Omron CX-Programmer project NewProject (CX-Programmer 9.61)

# PLC NewPLC1: CP1H X

## Global symbols (name address type ; comment)
0.00 BOOL  ; LIN3_FW
0.01 BOOL  ; EMG
0.02 BOOL  ; SY1
0.03 BOOL  ; CY1_FW
0.04 BOOL  ; CY1_BW
0.05 BOOL  ; CY2_A_1_BW
0.06 BOOL  ; CY2_A_2_BW
0.07 BOOL  ; CY3_FW
0.08 BOOL  ; CY3_BW
0.09 BOOL  ; CY4_A_1_BW
0.10 BOOL  ; CY4_A_2_BW
0.11 BOOL  ; S1_GRIPPER
100.00 BOOL  ; 1Y1
100.01 BOOL  ; 1Y2
100.02 BOOL  ; 2Y1
100.03 BOOL  ; 2Y2
100.04 BOOL  ; 4Y1
100.05 BOOL  ; 4Y2
100.06 BOOL  ; 3Y1
100.07 BOOL  ; 3Y2
101.00 BOOL  ; buzzzer
101.01 BOOL  ; ACTIVATE_SMC
101.02 BOOL  ; TRIGGER_MC2
101.03 BOOL  ; L_RED
101.04 BOOL  ; MOTOR_CONVEYOR
101.05 BOOL  ; TRIGGER RELAY
101.06 BOOL  ; ACTIVATE_MC2
102.00 BOOL  ; IN0 L1
102.01 BOOL  ; IN1 L1
102.02 BOOL  ; IN2 L1
102.03 BOOL  ; SETUP L1
102.04 BOOL  ; HOLD L1
102.05 BOOL  ; DRIVE L1
102.06 BOOL  ; RESET L1
102.07 BOOL  ; SVON L1
103.00 BOOL  ; IN0 L3
103.01 BOOL  ; IN1 L3
103.02 BOOL  ; IN2 L3
103.03 BOOL  ; SETUP L3
103.04 BOOL  ; HOLD L3
103.05 BOOL  ; DRIVE L3
103.06 BOOL  ; RESET L3
103.07 BOOL  ; SVON L3
104.00 BOOL  ; IN0 L2
104.01 BOOL  ; IN1 L2
104.02 BOOL  ; IN2 L2
104.03 BOOL  ; SETUP L2
104.04 BOOL  ; HOLD L2
104.05 BOOL  ; DRIVE L2
104.06 BOOL  ; RESET L2
104.07 BOOL  ; SVON L2
105.00 BOOL  ; C1
1500.00 BOOL  ; memory
1.00 BOOL  ; SL_LOADING
1.01 BOOL  ; SUL_UNLOADING
1.02 BOOL  ; LIN2_FW
1.03 BOOL  ; LIN3_BW
1.04 BOOL  ; LIN1_FW
1.05 BOOL  ; START1_CONV
1.06 BOOL  ; START2_CONV
1.07 BOOL  ; EMG_CONV
1.08 BOOL  ; SENSOR_CONV
1.09 BOOL  ; S2_GRIPPER
2000.00 BOOL  ; STEP0
2000.01 BOOL  ; STEP1
2000.02 BOOL  ; STEP2
2000.03 BOOL  ; STEP3
2000.04 BOOL  ; STEP4
2000.05 BOOL  ; STEP5
2000.06 BOOL  ; STEP6
2000.07 BOOL  ; STEP7
2000.08 BOOL  ; STEP8
2000.09 BOOL  ; STEP9
2000.10 BOOL  ; STEP10
2000.11 BOOL  ; STEP11
2000.12 BOOL  ; STEP12
2000.13 BOOL  ; STEP13
2000.14 BOOL  ; STEP14
2000.15 BOOL  ; STEP15
2001.00 BOOL  ; STEP1_2
2002.00 BOOL  ; STEP16
2002.01 BOOL  ; STEP17
2002.02 BOOL  ; STEP18
2002.03 BOOL  ; STEP19
2002.04 BOOL  ; STEP20
200.01 BOOL  ; HMI-PON
200.02 BOOL  ; HMI-POFF
200.03 BOOL  ; HMI-INIT
200.06 BOOL  ; START SIG AUTO
200.07 BOOL  ; STOP SIG AUTO
200.10 BOOL  ; fast
200.11 BOOL  ; RESET_LINEAR
201.00 BOOL  ; LIN_ON
201.01 BOOL  ; INIT LIN1
201.02 BOOL  ; LIN EMG OK
201.03 BOOL  ; LIN_ALM_OK
201.04 BOOL  ; INIT LIN2
201.05 BOOL  ; INIT LIN3
201.06 BOOL  ; INIT_CYL
201.07 BOOL  ; CYL_GRIP_INPOS
201.08 BOOL  ; CYL3_INPOS
201.09 BOOL  ; CYL1_INPOS
201.10 BOOL  ; INIT_CYL)OK
201.11 BOOL  ; INIT LIN OK
201.12 BOOL  ; Trigger_Auto
201.13 BOOL  ; AUTOSIG
201.14 BOOL  ; INIT OK
202.00 BOOL  ; LIN_1_Forward
202.01 BOOL  ; LIN_1_Backward
22.15 BOOL  ; MAIN_OK
2.00 BOOL  ; OUT1_L1
2.01 BOOL  ; OUT2_L1
2.02 BOOL  ; BUSY_L1
2.03 BOOL  ; SETON_L1
2.04 BOOL  ; INP_L1
2.05 BOOL  ; SVRE_L1
2.06 BOOL  ; ESTOP_L1
2.07 BOOL  ; ALARM_L1
3000.00 BOOL  ; STEP0
3000.01 BOOL  ; STEP1
3000.02 BOOL  ; STEP2
3000.03 BOOL  ; STEP3
3000.04 BOOL  ; STEP4
3000.05 BOOL  ; STEP5
3000.06 BOOL  ; STEP6
3000.07 BOOL  ; STEP7
3000.08 BOOL  ; STEP8
3000.09 BOOL  ; STEP9
3000.10 BOOL  ; STEP10
3000.11 BOOL  ; STEP11
300.00 BOOL  ; L1_LW
300.01 BOOL  ; L2 FW
300.02 BOOL  ; L3_FW1
300.03 BOOL  ; L3_FW2
300.04 BOOL  ; MAN_CY1_FW
300.05 BOOL  ; MAN_CY2_FW
300.06 BOOL  ; MAN_CY3_FW
300.07 BOOL  ; MAN_CY4_FW
300.08 BOOL  ; L1_MAN_BW
300.11 BOOL  ; L1_MAN_FW
30.00 BOOL  ; TIM_CONV
30.01 BOOL  ; LOCK_TIM
330.00 BOOL  ; MAN_L1_P1
330.01 BOOL  ; MAN_L1_P2
330.02 BOOL  ; MAN_L2_P1
330.03 BOOL  ; MAN_L2_P2
330.04 BOOL  ; MAN_L1_P1
330.05 BOOL  ; MAN_L1_P2
350.14 BOOL  ; Alarm_EMG
350.15 BOOL  ; Alarm_Main_Air_Supply
351.00 BOOL  ; Alarm_Lin1_OFF
351.01 BOOL  ; Alarm_Lin3_OFF
351.02 BOOL  ; Alarm_Lin2_OFF
351.03 BOOL  ; Alarm_SMC1
351.04 BOOL  ; Alarm_SMC3
351.05 BOOL  ; Alarm_SMC2
3.00 BOOL  ; OUT1_L3
3.01 BOOL  ; OUT2_L3
3.02 BOOL  ; BUSY_L3
3.03 BOOL  ; SETON_L3
3.04 BOOL  ; INP_L3
3.05 BOOL  ; SVRE_L3
3.06 BOOL  ; ESTOP_L3
3.07 BOOL  ; ALARM_L3
4000.00 BOOL  ; STEP0
4000.01 BOOL  ; STEP1
4000.02 BOOL  ; STEP2
4000.03 BOOL  ; STEP3
4000.04 BOOL  ; picking_alert
400.02 BOOL  ; Timer_homing
4.00 BOOL  ; OUT1_L2
4.01 BOOL  ; OUT2_L2
4.02 BOOL  ; BUSY_L2
4.03 BOOL  ; SETON_L2
4.04 BOOL  ; INPT_L2
4.05 BOOL  ; SVRE_L2
4.06 BOOL  ; ESTOP_L2
4.07 BOOL  ; ALARM_L2
600.00 BOOL  ; L1_BW
600.01 BOOL  ; LW_BW
600.02 BOOL  ; L3_BW
600.03 BOOL  ; CY1_BW
600.04 BOOL  ; MAN_CY1_BW
600.05 BOOL  ; MAN_CY2_BW
600.06 BOOL  ; MAN_CY3_BW
600.07 BOOL  ; MAN_CY4_BW
60.00 BOOL  ; DIFD_BUSY_L1
60.01 BOOL  ; DIFD_BUSY_L3
60.02 BOOL  ; DIFD_BUSY_L2
60.03 BOOL  ; DIFU_BUSY_L1
60.04 BOOL  ; DIFU_BUSY_L3
60.05 BOOL  ; DIFU_BUSY_L2
700.00 BOOL  ; L1 MAN GO
700.01 BOOL  ; L2 MAN GO
700.02 BOOL  ; L3 MAN GO
800.00 BOOL  ; AUTO/MAN
T0000 BOOL  ; TIM_S0
T0001 BOOL  ; TIM_S1
T0002 BOOL  ; TIM_S2
T0003 BOOL  ; TIM_S3
T0004 BOOL  ; TIM_S4
T0005 BOOL  ; TIM_S5
T0006 BOOL  ; TIM_S6
T0007 BOOL  ; TIM_S7
T0008 BOOL  ; TIM_S8
T0009 BOOL  ; TIM_S9
T0010 BOOL  ; TIM-S10
T0011 BOOL  ; TIM_S11
T0012 BOOL  ; TIM_S12
T0013 BOOL  ; TIM_S13
T0014 BOOL  ; TIM-S14
T0015 BOOL  ; TIM_STEP15
T0017 BOOL  ; TIM_S17
T0018 BOOL  ; TIM_S18
T0019 BOOL  ; TIM_S19
T0030 BOOL  ; T-S0
T0031 BOOL  ; T-S1
T0032 BOOL  ; T-S2
T0033 BOOL  ; T-S3
T0034 BOOL  ; T-S4
T0035 BOOL  ; t-S5
T0036 BOOL  ; T-S6
T0037 BOOL  ; STEP7
T0038 BOOL  ; T-S8
T0039 BOOL  ; t-S9
T0040 BOOL  ; T-S10
T0050 BOOL  ; T-S0
T0051 BOOL  ; T-S1
T0052 BOOL  ; t-s2
T0070 BOOL  ; timer delay turun
T0071 BOOL  ; Delay gerak maju
T0200 BOOL  ; TIMS1_CONV
T0201 BOOL  ; TIMS2_CONV
T0202 BOOL  ; TIM_PRESENCE
T0203 BOOL  ; L1_MAN_TIM
T0420 BOOL  ; Timer Trigger Position auto
T1000 BOOL  ; TIM_S1_2

## Program NewProgram1 (cyclic task 0)
; CONVEYOR EVACUATION

### Section INIT_MAIN

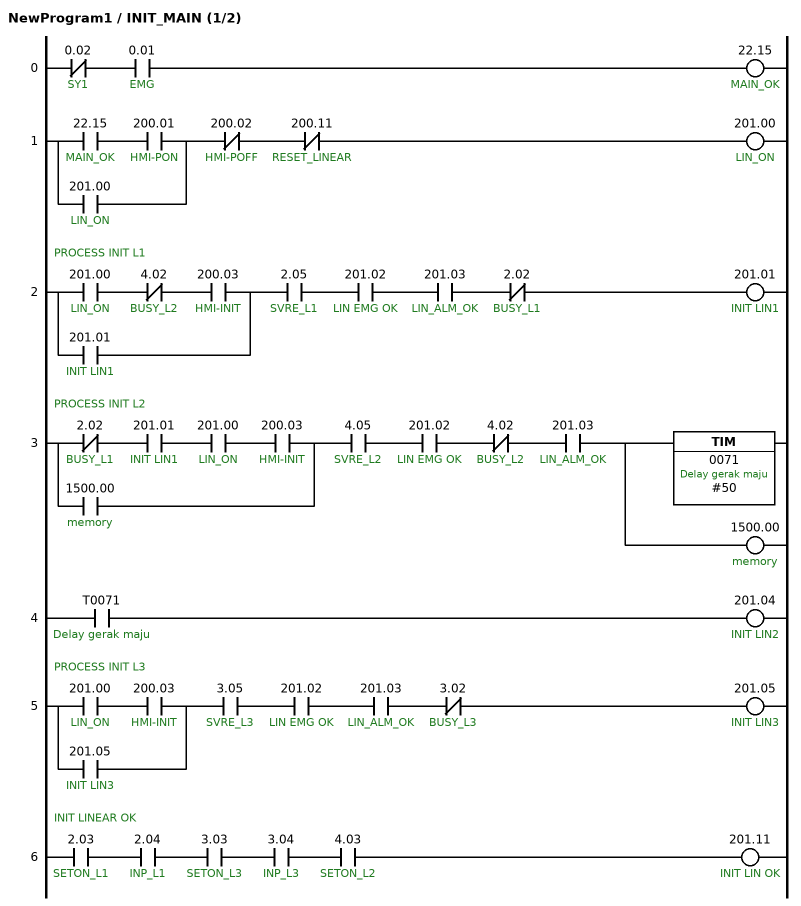
; rung 0
LDNOT 0.02  ; SY1
AND 0.01  ; EMG
OUT 22.15  ; MAIN_OK
; rung 1
LD 22.15  ; MAIN_OK
AND 200.01  ; HMI-PON
OR 201.00  ; LIN_ON
ANDNOT 200.02  ; HMI-POFF
ANDNOT 200.11  ; RESET_LINEAR
OUT 201.00  ; LIN_ON
; rung 2: PROCESS INIT L1
LD 201.00  ; LIN_ON
ANDNOT 4.02  ; BUSY_L2  // tambahan santo
AND 200.03  ; HMI-INIT
OR 201.01  ; INIT LIN1
AND 2.05  ; SVRE_L1
AND 201.02  ; LIN EMG OK
AND 201.03  ; LIN_ALM_OK
ANDNOT 2.02  ; BUSY_L1
OUT 201.01  ; INIT LIN1
; rung 3: PROCESS INIT L2
LDNOT 2.02  ; BUSY_L1  // tambahan santo
AND 201.01  ; INIT LIN1  // Tambahan santo
AND 201.00  ; LIN_ON
AND 200.03  ; HMI-INIT
OR 1500.00  ; memory
AND 4.05  ; SVRE_L2
AND 201.02  ; LIN EMG OK
ANDNOT 4.02  ; BUSY_L2
AND 201.03  ; LIN_ALM_OK
TIM 0071 #50  ; Delay gerak maju
OUT 1500.00  ; memory
; rung 4
LD T0071  ; Delay gerak maju
OUT 201.04  ; INIT LIN2
; rung 5: PROCESS INIT L3
LD 201.00  ; LIN_ON
AND 200.03  ; HMI-INIT
OR 201.05  ; INIT LIN3
AND 3.05  ; SVRE_L3
AND 201.02  ; LIN EMG OK
AND 201.03  ; LIN_ALM_OK
ANDNOT 3.02  ; BUSY_L3
OUT 201.05  ; INIT LIN3
; rung 6: INIT LINEAR OK
LD 2.03  ; SETON_L1
AND 2.04  ; INP_L1
AND 3.03  ; SETON_L3
AND 3.04  ; INP_L3
AND 4.03  ; SETON_L2
OUT 201.11  ; INIT LIN OK

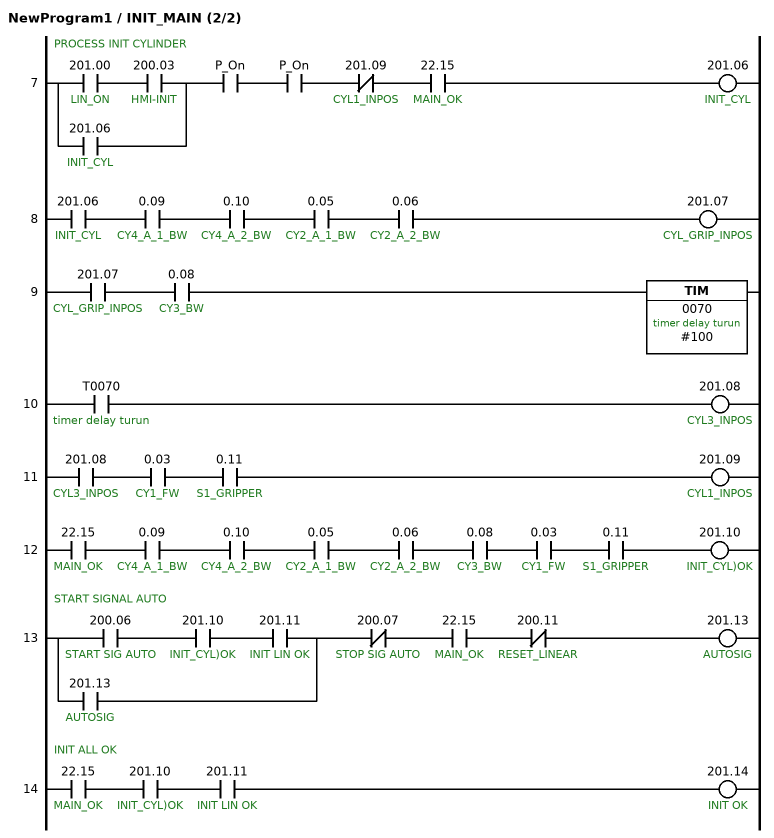
; rung 7: PROCESS INIT CYLINDER
LD 201.00  ; LIN_ON
AND 200.03  ; HMI-INIT
OR 201.06  ; INIT_CYL
AND P_On
AND P_On
ANDNOT 201.09  ; CYL1_INPOS
AND 22.15  ; MAIN_OK
OUT 201.06  ; INIT_CYL
; rung 8
LD 201.06  ; INIT_CYL
AND 0.09  ; CY4_A_1_BW
AND 0.10  ; CY4_A_2_BW
AND 0.05  ; CY2_A_1_BW
AND 0.06  ; CY2_A_2_BW
OUT 201.07  ; CYL_GRIP_INPOS
; rung 9
LD 201.07  ; CYL_GRIP_INPOS
AND 0.08  ; CY3_BW
TIM 0070 #100  ; timer delay turun
; rung 10
LD T0070  ; timer delay turun
OUT 201.08  ; CYL3_INPOS
; rung 11
LD 201.08  ; CYL3_INPOS
AND 0.03  ; CY1_FW
AND 0.11  ; S1_GRIPPER
OUT 201.09  ; CYL1_INPOS
; rung 12
LD 22.15  ; MAIN_OK
AND 0.09  ; CY4_A_1_BW
AND 0.10  ; CY4_A_2_BW
AND 0.05  ; CY2_A_1_BW
AND 0.06  ; CY2_A_2_BW
AND 0.08  ; CY3_BW
AND 0.03  ; CY1_FW
AND 0.11  ; S1_GRIPPER
OUT 201.10  ; INIT_CYL)OK
; rung 13: START SIGNAL AUTO
LD 200.06  ; START SIG AUTO
AND 201.10  ; INIT_CYL)OK
AND 201.11  ; INIT LIN OK
OR 201.13  ; AUTOSIG
ANDNOT 200.07  ; STOP SIG AUTO
AND 22.15  ; MAIN_OK
ANDNOT 200.11  ; RESET_LINEAR
OUT 201.13  ; AUTOSIG
; rung 14: INIT ALL OK
LD 22.15  ; MAIN_OK
AND 201.10  ; INIT_CYL)OK
AND 201.11  ; INIT LIN OK
OUT 201.14  ; INIT OK

### Section ALARM

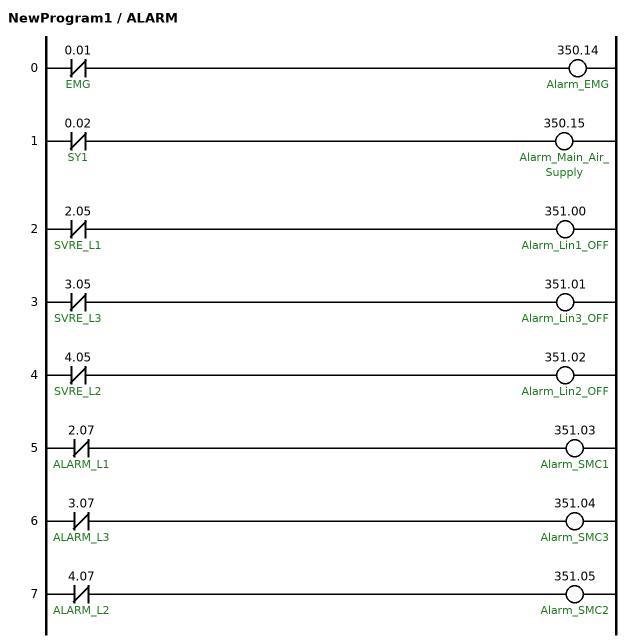
; rung 0
LDNOT 0.01  ; EMG
OUT 350.14  ; Alarm_EMG
; rung 1
LDNOT 0.02  ; SY1
OUT 350.15  ; Alarm_Main_Air_Supply
; rung 2
LDNOT 2.05  ; SVRE_L1
OUT 351.00  ; Alarm_Lin1_OFF
; rung 3
LDNOT 3.05  ; SVRE_L3
OUT 351.01  ; Alarm_Lin3_OFF
; rung 4
LDNOT 4.05  ; SVRE_L2
OUT 351.02  ; Alarm_Lin2_OFF
; rung 5
LDNOT 2.07  ; ALARM_L1
OUT 351.03  ; Alarm_SMC1
; rung 6
LDNOT 3.07  ; ALARM_L3
OUT 351.04  ; Alarm_SMC3
; rung 7
LDNOT 4.07  ; ALARM_L2
OUT 351.05  ; Alarm_SMC2

### Section LINEAR_CONTROL_OUT

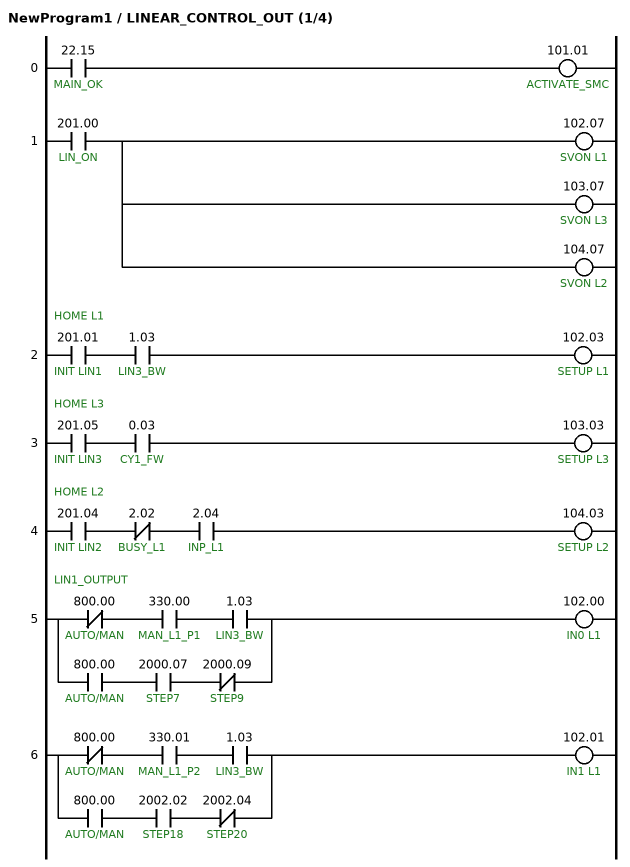
; rung 0
LD 22.15  ; MAIN_OK
OUT 101.01  ; ACTIVATE_SMC
; rung 1
LD 201.00  ; LIN_ON
OUT 102.07  ; SVON L1
OUT 103.07  ; SVON L3
OUT 104.07  ; SVON L2
; rung 2: HOME L1
LD 201.01  ; INIT LIN1
AND 1.03  ; LIN3_BW
OUT 102.03  ; SETUP L1
; rung 3: HOME L3
LD 201.05  ; INIT LIN3
AND 0.03  ; CY1_FW
OUT 103.03  ; SETUP L3
; rung 4: HOME L2
LD 201.04  ; INIT LIN2
ANDNOT 2.02  ; BUSY_L1
AND 2.04  ; INP_L1
OUT 104.03  ; SETUP L2
; rung 5: LIN1_OUTPUT
LDNOT 800.00  ; AUTO/MAN
AND 330.00  ; MAN_L1_P1
AND 1.03  ; LIN3_BW
LD 800.00  ; AUTO/MAN
AND 2000.07  ; STEP7
ANDNOT 2000.09  ; STEP9
ORLD
OUT 102.00  ; IN0 L1
; rung 6
LDNOT 800.00  ; AUTO/MAN
AND 330.01  ; MAN_L1_P2
AND 1.03  ; LIN3_BW
LD 800.00  ; AUTO/MAN
AND 2002.02  ; STEP18
ANDNOT 2002.04  ; STEP20
ORLD
OUT 102.01  ; IN1 L1

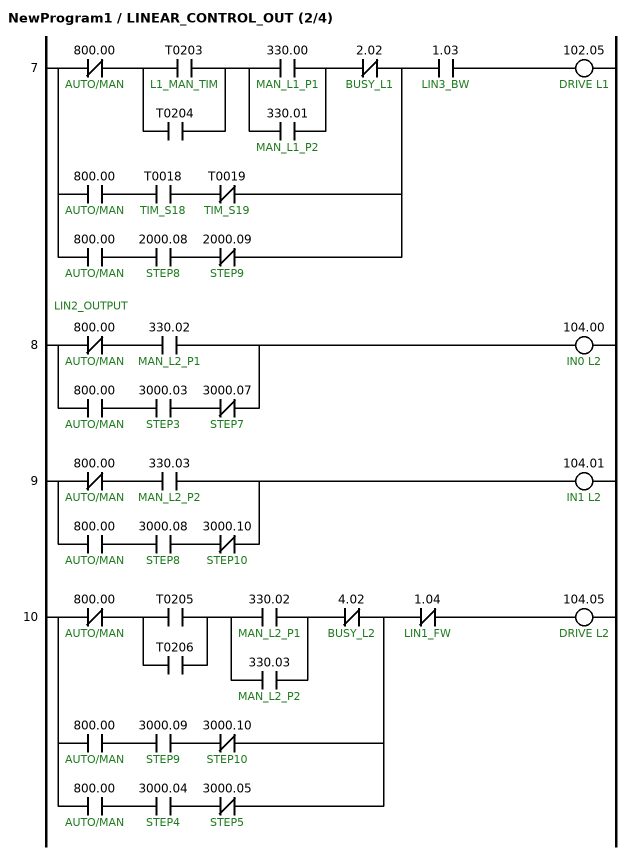
; rung 7
LDNOT 800.00  ; AUTO/MAN
LD T0203  ; L1_MAN_TIM
OR T0204
ANDLD
LD 330.00  ; MAN_L1_P1
OR 330.01  ; MAN_L1_P2
ANDLD
ANDNOT 2.02  ; BUSY_L1
LD 800.00  ; AUTO/MAN
AND T0018  ; TIM_S18
ANDNOT T0019  ; TIM_S19
ORLD
LD 800.00  ; AUTO/MAN
AND 2000.08  ; STEP8
ANDNOT 2000.09  ; STEP9
ORLD
AND 1.03  ; LIN3_BW
OUT 102.05  ; DRIVE L1
; rung 8: LIN2_OUTPUT
LDNOT 800.00  ; AUTO/MAN
AND 330.02  ; MAN_L2_P1
LD 800.00  ; AUTO/MAN
AND 3000.03  ; STEP3
ANDNOT 3000.07  ; STEP7
ORLD
OUT 104.00  ; IN0 L2
; rung 9
LDNOT 800.00  ; AUTO/MAN
AND 330.03  ; MAN_L2_P2
LD 800.00  ; AUTO/MAN
AND 3000.08  ; STEP8
ANDNOT 3000.10  ; STEP10
ORLD
OUT 104.01  ; IN1 L2
; rung 10
LDNOT 800.00  ; AUTO/MAN
LD T0205
OR T0206
ANDLD
LD 330.02  ; MAN_L2_P1
OR 330.03  ; MAN_L2_P2
ANDLD
ANDNOT 4.02  ; BUSY_L2
LD 800.00  ; AUTO/MAN
AND 3000.09  ; STEP9
ANDNOT 3000.10  ; STEP10
ORLD
LD 800.00  ; AUTO/MAN
AND 3000.04  ; STEP4
ANDNOT 3000.05  ; STEP5
ORLD
ANDNOT 1.04  ; LIN1_FW
OUT 104.05  ; DRIVE L2

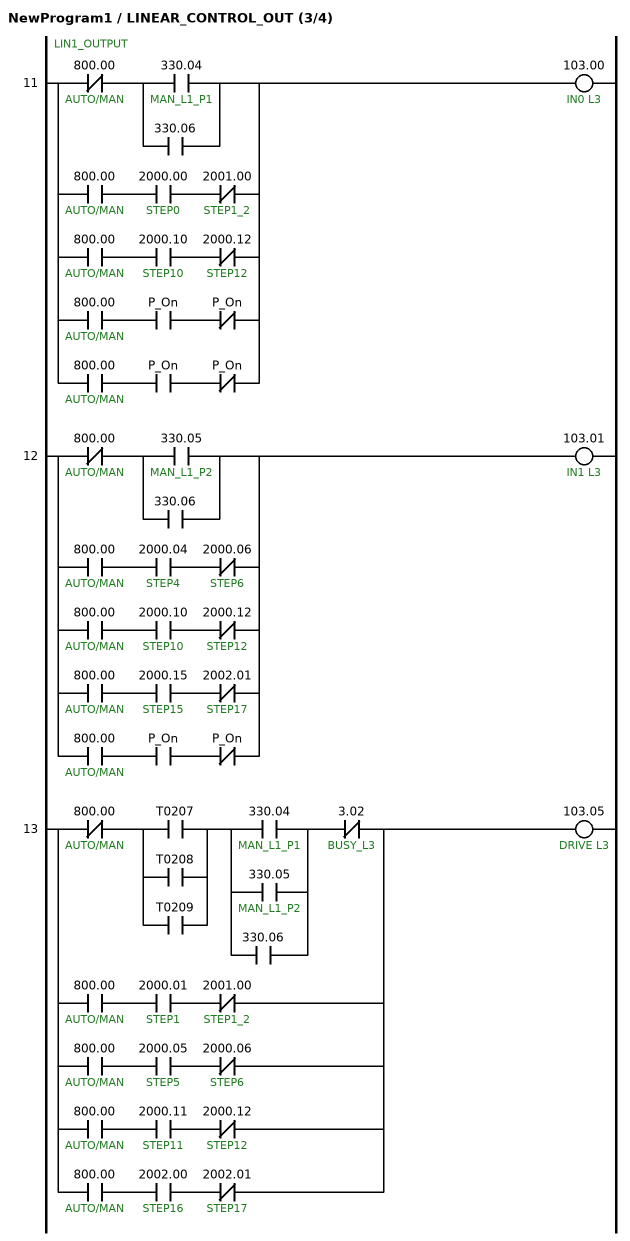
; rung 11: LIN1_OUTPUT
LDNOT 800.00  ; AUTO/MAN
LD 330.04  ; MAN_L1_P1
OR 330.06
ANDLD
LD 800.00  ; AUTO/MAN
AND 2000.00  ; STEP0
ANDNOT 2001.00  ; STEP1_2
ORLD
LD 800.00  ; AUTO/MAN
AND 2000.10  ; STEP10
ANDNOT 2000.12  ; STEP12
ORLD
LD 800.00  ; AUTO/MAN
AND P_On
ANDNOT P_On
ORLD
LD 800.00  ; AUTO/MAN
AND P_On
ANDNOT P_On
ORLD
OUT 103.00  ; IN0 L3
; rung 12
LDNOT 800.00  ; AUTO/MAN
LD 330.05  ; MAN_L1_P2
OR 330.06
ANDLD
LD 800.00  ; AUTO/MAN
AND 2000.04  ; STEP4
ANDNOT 2000.06  ; STEP6
ORLD
LD 800.00  ; AUTO/MAN
AND 2000.10  ; STEP10
ANDNOT 2000.12  ; STEP12
ORLD
LD 800.00  ; AUTO/MAN
AND 2000.15  ; STEP15
ANDNOT 2002.01  ; STEP17
ORLD
LD 800.00  ; AUTO/MAN
AND P_On
ANDNOT P_On
ORLD
OUT 103.01  ; IN1 L3
; rung 13
LDNOT 800.00  ; AUTO/MAN
LD T0207
OR T0208
OR T0209
ANDLD
LD 330.04  ; MAN_L1_P1
OR 330.05  ; MAN_L1_P2
OR 330.06
ANDLD
ANDNOT 3.02  ; BUSY_L3
LD 800.00  ; AUTO/MAN
AND 2000.01  ; STEP1
ANDNOT 2001.00  ; STEP1_2
ORLD
LD 800.00  ; AUTO/MAN
AND 2000.05  ; STEP5
ANDNOT 2000.06  ; STEP6
ORLD
LD 800.00  ; AUTO/MAN
AND 2000.11  ; STEP11
ANDNOT 2000.12  ; STEP12
ORLD
LD 800.00  ; AUTO/MAN
AND 2002.00  ; STEP16
ANDNOT 2002.01  ; STEP17
ORLD
OUT 103.05  ; DRIVE L3

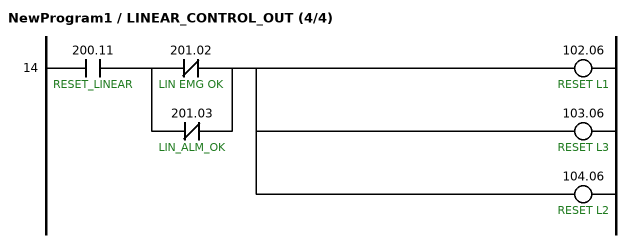
; rung 14
LD 200.11  ; RESET_LINEAR
LDNOT 201.02  ; LIN EMG OK
ORNOT 201.03  ; LIN_ALM_OK
ANDLD
OUT 102.06  ; RESET L1
OUT 103.06  ; RESET L3
OUT 104.06  ; RESET L2

### Section CYLINDER_CONTROL_OUT

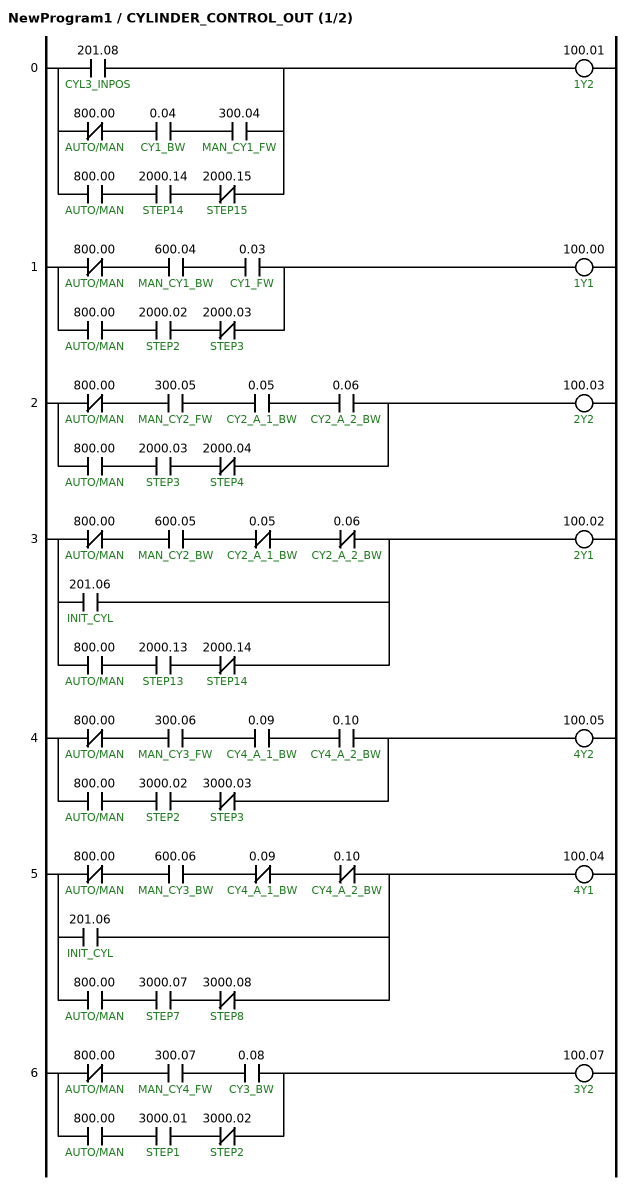
; rung 0
LD 201.08  ; CYL3_INPOS
LDNOT 800.00  ; AUTO/MAN
AND 0.04  ; CY1_BW
AND 300.04  ; MAN_CY1_FW
ORLD
LD 800.00  ; AUTO/MAN
AND 2000.14  ; STEP14
ANDNOT 2000.15  ; STEP15
ORLD
OUT 100.01  ; 1Y2
; rung 1
LDNOT 800.00  ; AUTO/MAN
AND 600.04  ; MAN_CY1_BW
AND 0.03  ; CY1_FW
LD 800.00  ; AUTO/MAN
AND 2000.02  ; STEP2
ANDNOT 2000.03  ; STEP3
ORLD
OUT 100.00  ; 1Y1
; rung 2
LDNOT 800.00  ; AUTO/MAN
AND 300.05  ; MAN_CY2_FW
AND 0.05  ; CY2_A_1_BW
AND 0.06  ; CY2_A_2_BW
LD 800.00  ; AUTO/MAN
AND 2000.03  ; STEP3
ANDNOT 2000.04  ; STEP4
ORLD
OUT 100.03  ; 2Y2
; rung 3
LDNOT 800.00  ; AUTO/MAN
AND 600.05  ; MAN_CY2_BW
ANDNOT 0.05  ; CY2_A_1_BW
ANDNOT 0.06  ; CY2_A_2_BW
OR 201.06  ; INIT_CYL
LD 800.00  ; AUTO/MAN
AND 2000.13  ; STEP13
ANDNOT 2000.14  ; STEP14
ORLD
OUT 100.02  ; 2Y1
; rung 4
LDNOT 800.00  ; AUTO/MAN
AND 300.06  ; MAN_CY3_FW
AND 0.09  ; CY4_A_1_BW
AND 0.10  ; CY4_A_2_BW
LD 800.00  ; AUTO/MAN
AND 3000.02  ; STEP2
ANDNOT 3000.03  ; STEP3
ORLD
OUT 100.05  ; 4Y2
; rung 5
LDNOT 800.00  ; AUTO/MAN
AND 600.06  ; MAN_CY3_BW
ANDNOT 0.09  ; CY4_A_1_BW
ANDNOT 0.10  ; CY4_A_2_BW
OR 201.06  ; INIT_CYL
LD 800.00  ; AUTO/MAN
AND 3000.07  ; STEP7
ANDNOT 3000.08  ; STEP8
ORLD
OUT 100.04  ; 4Y1
; rung 6
LDNOT 800.00  ; AUTO/MAN
AND 300.07  ; MAN_CY4_FW
AND 0.08  ; CY3_BW
LD 800.00  ; AUTO/MAN
AND 3000.01  ; STEP1
ANDNOT 3000.02  ; STEP2
ORLD
OUT 100.07  ; 3Y2

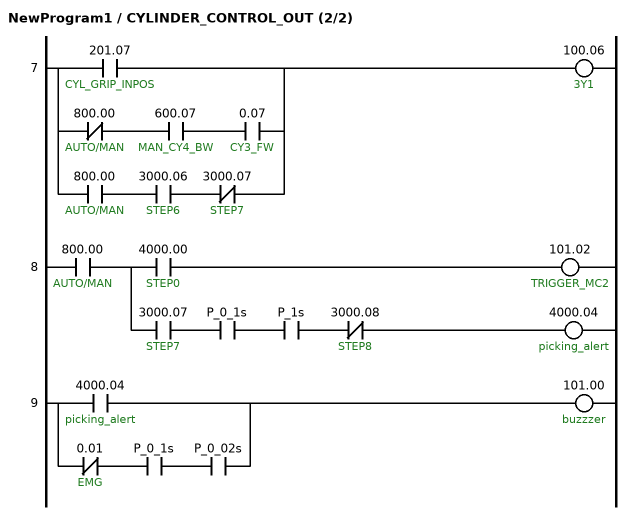
; rung 7
LD 201.07  ; CYL_GRIP_INPOS
LDNOT 800.00  ; AUTO/MAN
AND 600.07  ; MAN_CY4_BW
AND 0.07  ; CY3_FW
ORLD
LD 800.00  ; AUTO/MAN
AND 3000.06  ; STEP6
ANDNOT 3000.07  ; STEP7
ORLD
OUT 100.06  ; 3Y1
; rung 8
LD 800.00  ; AUTO/MAN
OUT TR0
AND 4000.00  ; STEP0
OUT 101.02  ; TRIGGER_MC2
LD TR0
AND 3000.07  ; STEP7
AND P_0_1s
AND P_1s
ANDNOT 3000.08  ; STEP8
OUT 4000.04  ; picking_alert
; rung 9
LD 4000.04  ; picking_alert
LDNOT 0.01  ; EMG
AND P_0_1s
AND P_0_02s
ORLD
OUT 101.00  ; buzzzer

### Section LINEAR_DATA_STATUS

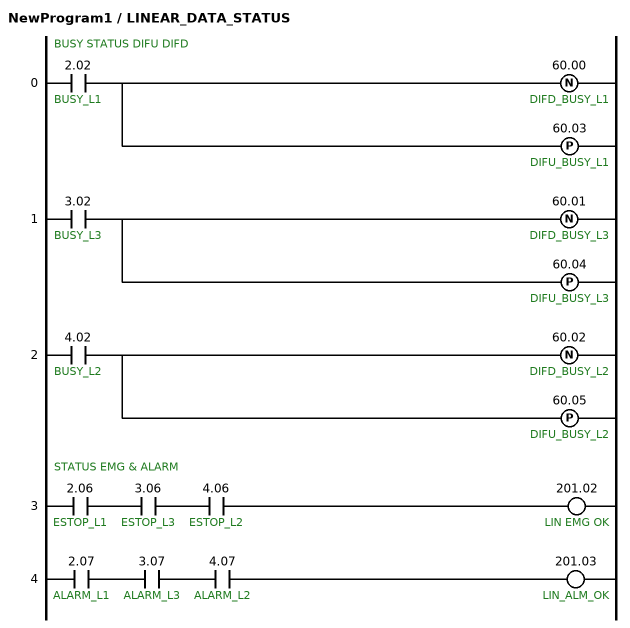
; rung 0: BUSY STATUS DIFU DIFD
LD 2.02  ; BUSY_L1
DIFD(014) 60.00  ; DIFD_BUSY_L1
DIFU(013) 60.03  ; DIFU_BUSY_L1
; rung 1
LD 3.02  ; BUSY_L3
DIFD(014) 60.01  ; DIFD_BUSY_L3
DIFU(013) 60.04  ; DIFU_BUSY_L3
; rung 2
LD 4.02  ; BUSY_L2
DIFD(014) 60.02  ; DIFD_BUSY_L2
DIFU(013) 60.05  ; DIFU_BUSY_L2
; rung 3: STATUS EMG & ALARM
LD 2.06  ; ESTOP_L1
AND 3.06  ; ESTOP_L3
AND 4.06  ; ESTOP_L2
OUT 201.02  ; LIN EMG OK
; rung 4
LD 2.07  ; ALARM_L1
AND 3.07  ; ALARM_L3
AND 4.07  ; ALARM_L2
OUT 201.03  ; LIN_ALM_OK

### Section LINEAR_MANUAL

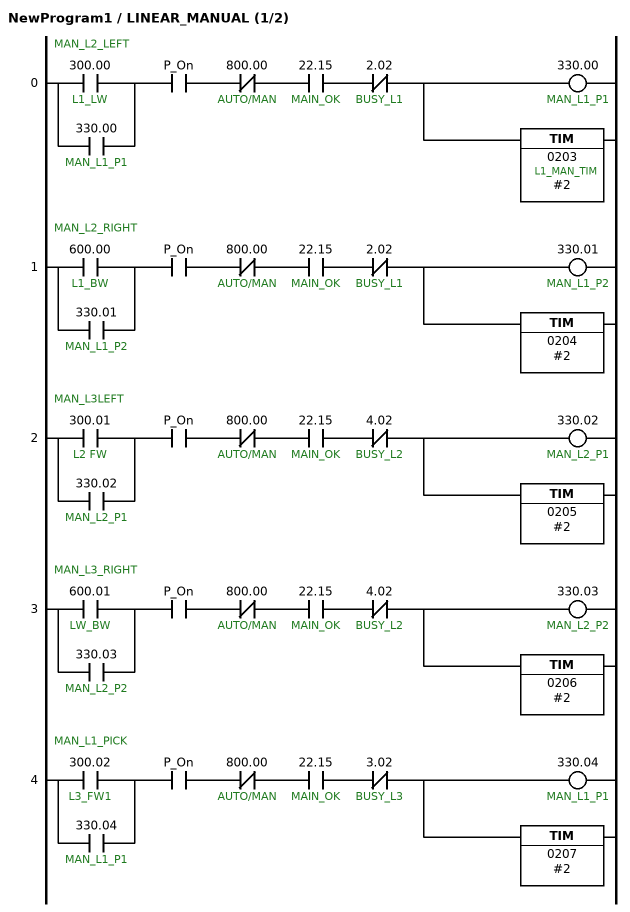
; rung 0: MAN_L2_LEFT
LD 300.00  ; L1_LW
OR 330.00  ; MAN_L1_P1
AND P_On
ANDNOT 800.00  ; AUTO/MAN
AND 22.15  ; MAIN_OK
ANDNOT 2.02  ; BUSY_L1
OUT 330.00  ; MAN_L1_P1
TIM 0203 #2  ; L1_MAN_TIM
; rung 1: MAN_L2_RIGHT
LD 600.00  ; L1_BW
OR 330.01  ; MAN_L1_P2
AND P_On
ANDNOT 800.00  ; AUTO/MAN
AND 22.15  ; MAIN_OK
ANDNOT 2.02  ; BUSY_L1
OUT 330.01  ; MAN_L1_P2
TIM 0204 #2
; rung 2: MAN_L3LEFT
LD 300.01  ; L2 FW
OR 330.02  ; MAN_L2_P1
AND P_On
ANDNOT 800.00  ; AUTO/MAN
AND 22.15  ; MAIN_OK
ANDNOT 4.02  ; BUSY_L2
OUT 330.02  ; MAN_L2_P1
TIM 0205 #2
; rung 3: MAN_L3_RIGHT
LD 600.01  ; LW_BW
OR 330.03  ; MAN_L2_P2
AND P_On
ANDNOT 800.00  ; AUTO/MAN
AND 22.15  ; MAIN_OK
ANDNOT 4.02  ; BUSY_L2
OUT 330.03  ; MAN_L2_P2
TIM 0206 #2
; rung 4: MAN_L1_PICK
LD 300.02  ; L3_FW1
OR 330.04  ; MAN_L1_P1
AND P_On
ANDNOT 800.00  ; AUTO/MAN
AND 22.15  ; MAIN_OK
ANDNOT 3.02  ; BUSY_L3
OUT 330.04  ; MAN_L1_P1
TIM 0207 #2

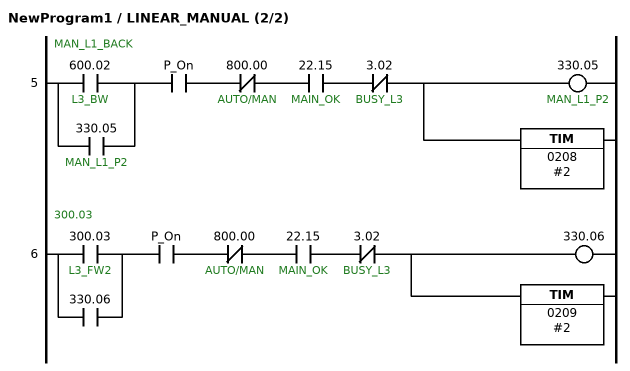
; rung 5: MAN_L1_BACK
LD 600.02  ; L3_BW
OR 330.05  ; MAN_L1_P2
AND P_On
ANDNOT 800.00  ; AUTO/MAN
AND 22.15  ; MAIN_OK
ANDNOT 3.02  ; BUSY_L3
OUT 330.05  ; MAN_L1_P2
TIM 0208 #2
; rung 6: 300.03
LD 300.03  ; L3_FW2
OR 330.06
AND P_On
ANDNOT 800.00  ; AUTO/MAN
AND 22.15  ; MAIN_OK
ANDNOT 3.02  ; BUSY_L3
OUT 330.06
TIM 0209 #2

### Section SEQUENCE_SECTION1

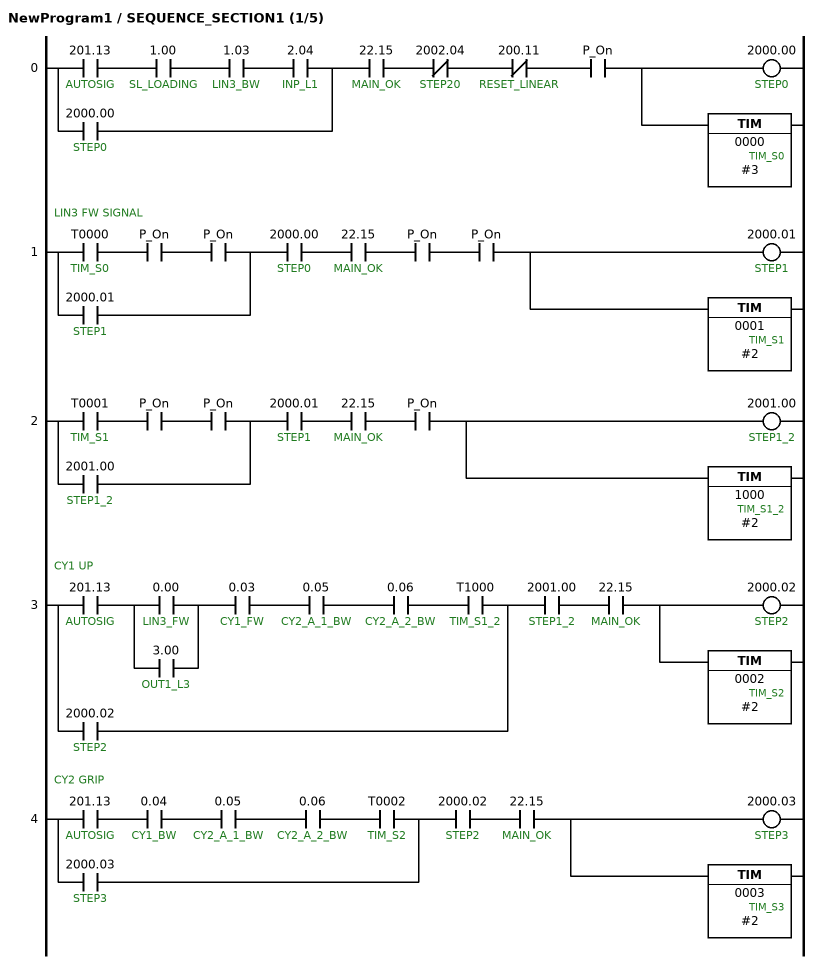
; rung 0
LD 201.13  ; AUTOSIG
AND 1.00  ; SL_LOADING
AND 1.03  ; LIN3_BW
AND 2.04  ; INP_L1
OR 2000.00  ; STEP0
AND 22.15  ; MAIN_OK
ANDNOT 2002.04  ; STEP20
ANDNOT 200.11  ; RESET_LINEAR
AND P_On
OUT 2000.00  ; STEP0
TIM 0000 #3  ; TIM_S0
; rung 1: LIN3 FW SIGNAL
LD T0000  ; TIM_S0
AND P_On
AND P_On
OR 2000.01  ; STEP1
AND 2000.00  ; STEP0
AND 22.15  ; MAIN_OK
AND P_On
AND P_On
OUT 2000.01  ; STEP1
TIM 0001 #2  ; TIM_S1
; rung 2
LD T0001  ; TIM_S1
AND P_On
AND P_On
OR 2001.00  ; STEP1_2
AND 2000.01  ; STEP1
AND 22.15  ; MAIN_OK
AND P_On
OUT 2001.00  ; STEP1_2
TIM 1000 #2  ; TIM_S1_2
; rung 3: CY1 UP
LD 201.13  ; AUTOSIG
LD 0.00  ; LIN3_FW
OR 3.00  ; OUT1_L3
ANDLD
AND 0.03  ; CY1_FW
AND 0.05  ; CY2_A_1_BW
AND 0.06  ; CY2_A_2_BW
AND T1000  ; TIM_S1_2
OR 2000.02  ; STEP2
AND 2001.00  ; STEP1_2
AND 22.15  ; MAIN_OK
OUT 2000.02  ; STEP2
TIM 0002 #2  ; TIM_S2
; rung 4: CY2 GRIP
LD 201.13  ; AUTOSIG
AND 0.04  ; CY1_BW
AND 0.05  ; CY2_A_1_BW
AND 0.06  ; CY2_A_2_BW
AND T0002  ; TIM_S2
OR 2000.03  ; STEP3
AND 2000.02  ; STEP2
AND 22.15  ; MAIN_OK
OUT 2000.03  ; STEP3
TIM 0003 #2  ; TIM_S3

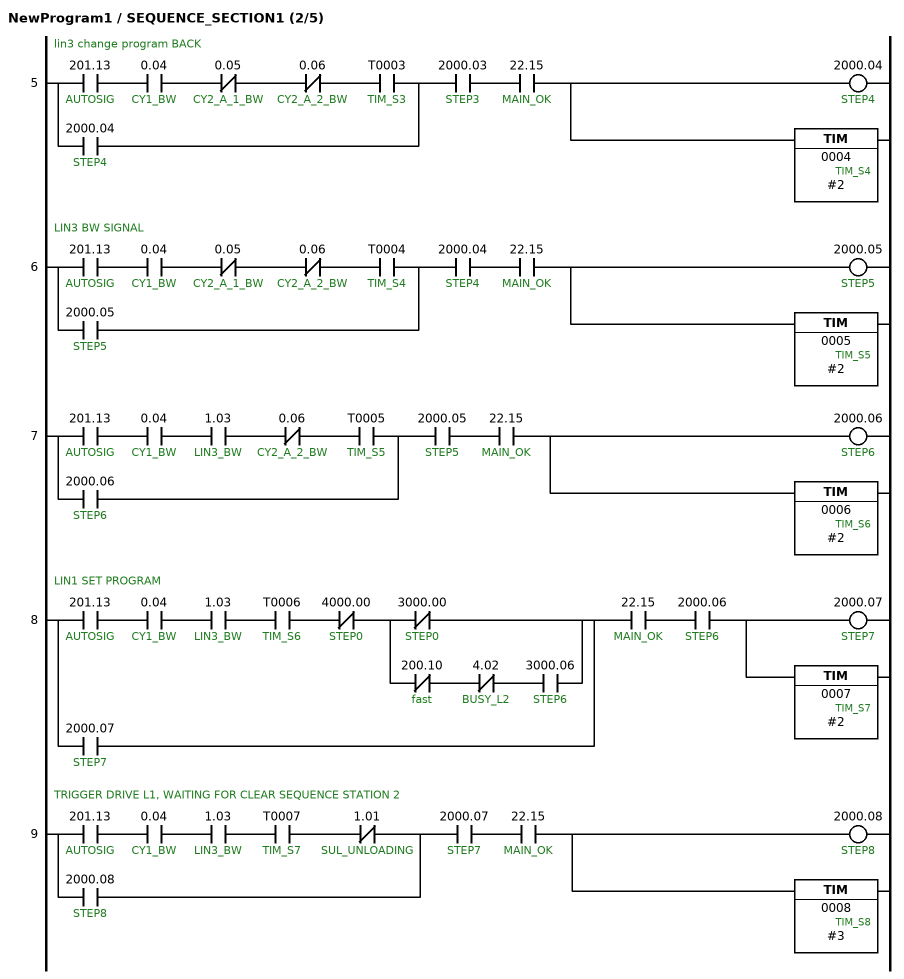
; rung 5: lin3 change program BACK
LD 201.13  ; AUTOSIG
AND 0.04  ; CY1_BW
ANDNOT 0.05  ; CY2_A_1_BW
ANDNOT 0.06  ; CY2_A_2_BW
AND T0003  ; TIM_S3
OR 2000.04  ; STEP4
AND 2000.03  ; STEP3
AND 22.15  ; MAIN_OK
OUT 2000.04  ; STEP4
TIM 0004 #2  ; TIM_S4
; rung 6: LIN3 BW SIGNAL
LD 201.13  ; AUTOSIG
AND 0.04  ; CY1_BW
ANDNOT 0.05  ; CY2_A_1_BW
ANDNOT 0.06  ; CY2_A_2_BW
AND T0004  ; TIM_S4
OR 2000.05  ; STEP5
AND 2000.04  ; STEP4
AND 22.15  ; MAIN_OK
OUT 2000.05  ; STEP5
TIM 0005 #2  ; TIM_S5
; rung 7
LD 201.13  ; AUTOSIG
AND 0.04  ; CY1_BW
AND 1.03  ; LIN3_BW
ANDNOT 0.06  ; CY2_A_2_BW
AND T0005  ; TIM_S5
OR 2000.06  ; STEP6
AND 2000.05  ; STEP5
AND 22.15  ; MAIN_OK
OUT 2000.06  ; STEP6
TIM 0006 #2  ; TIM_S6
; rung 8: LIN1 SET PROGRAM
LD 201.13  ; AUTOSIG
AND 0.04  ; CY1_BW
AND 1.03  ; LIN3_BW
AND T0006  ; TIM_S6
ANDNOT 4000.00  ; STEP0
LDNOT 3000.00  ; STEP0
LDNOT 200.10  ; fast
ANDNOT 4.02  ; BUSY_L2  // Tambahan santo
AND 3000.06  ; STEP6
ORLD
ANDLD
OR 2000.07  ; STEP7
AND 22.15  ; MAIN_OK
AND 2000.06  ; STEP6
OUT 2000.07  ; STEP7
TIM 0007 #2  ; TIM_S7
; rung 9: TRIGGER DRIVE L1, WAITING FOR CLEAR SEQUENCE STATION 2
LD 201.13  ; AUTOSIG
AND 0.04  ; CY1_BW
AND 1.03  ; LIN3_BW
AND T0007  ; TIM_S7
ANDNOT 1.01  ; SUL_UNLOADING
OR 2000.08  ; STEP8
AND 2000.07  ; STEP7
AND 22.15  ; MAIN_OK
OUT 2000.08  ; STEP8
TIM 0008 #3  ; TIM_S8

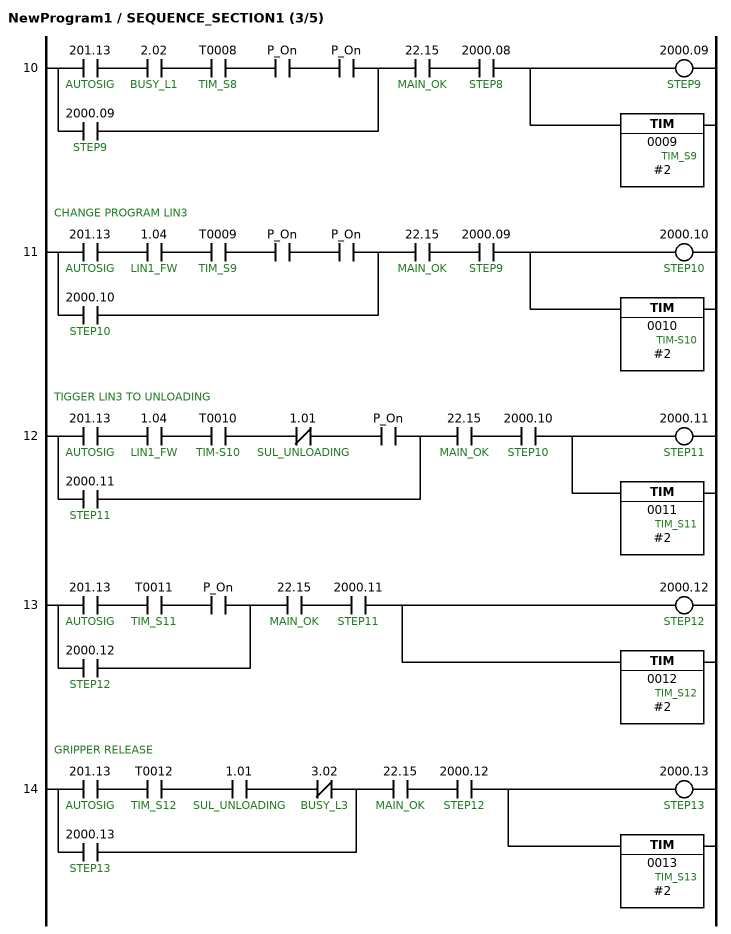
; rung 10
LD 201.13  ; AUTOSIG
AND 2.02  ; BUSY_L1
AND T0008  ; TIM_S8
AND P_On
AND P_On
OR 2000.09  ; STEP9
AND 22.15  ; MAIN_OK
AND 2000.08  ; STEP8
OUT 2000.09  ; STEP9
TIM 0009 #2  ; TIM_S9
; rung 11: CHANGE PROGRAM LIN3
LD 201.13  ; AUTOSIG
AND 1.04  ; LIN1_FW
AND T0009  ; TIM_S9
AND P_On
AND P_On
OR 2000.10  ; STEP10
AND 22.15  ; MAIN_OK
AND 2000.09  ; STEP9
OUT 2000.10  ; STEP10
TIM 0010 #2  ; TIM-S10
; rung 12: TIGGER LIN3 TO UNLOADING
LD 201.13  ; AUTOSIG
AND 1.04  ; LIN1_FW
AND T0010  ; TIM-S10
ANDNOT 1.01  ; SUL_UNLOADING
AND P_On
OR 2000.11  ; STEP11
AND 22.15  ; MAIN_OK
AND 2000.10  ; STEP10
OUT 2000.11  ; STEP11
TIM 0011 #2  ; TIM_S11
; rung 13
LD 201.13  ; AUTOSIG
AND T0011  ; TIM_S11
AND P_On
OR 2000.12  ; STEP12
AND 22.15  ; MAIN_OK
AND 2000.11  ; STEP11
OUT 2000.12  ; STEP12
TIM 0012 #2  ; TIM_S12
; rung 14: GRIPPER RELEASE
LD 201.13  ; AUTOSIG
AND T0012  ; TIM_S12
AND 1.01  ; SUL_UNLOADING
ANDNOT 3.02  ; BUSY_L3
OR 2000.13  ; STEP13
AND 22.15  ; MAIN_OK
AND 2000.12  ; STEP12
OUT 2000.13  ; STEP13
TIM 0013 #2  ; TIM_S13

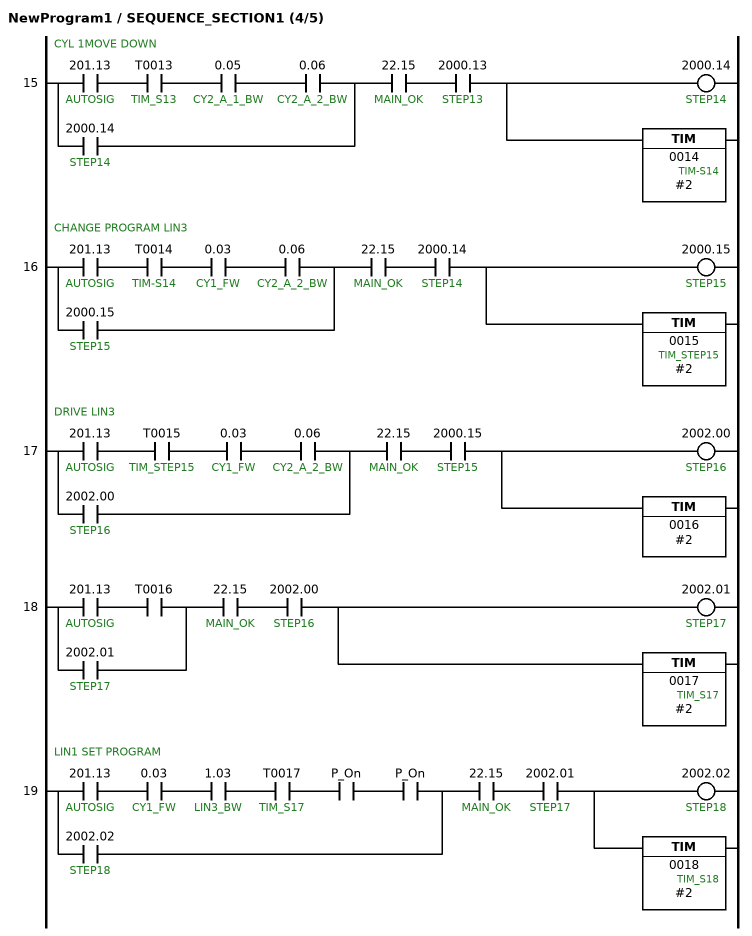
; rung 15: CYL 1MOVE DOWN
LD 201.13  ; AUTOSIG
AND T0013  ; TIM_S13
AND 0.05  ; CY2_A_1_BW
AND 0.06  ; CY2_A_2_BW
OR 2000.14  ; STEP14
AND 22.15  ; MAIN_OK
AND 2000.13  ; STEP13
OUT 2000.14  ; STEP14
TIM 0014 #2  ; TIM-S14
; rung 16: CHANGE PROGRAM LIN3
LD 201.13  ; AUTOSIG
AND T0014  ; TIM-S14
AND 0.03  ; CY1_FW
AND 0.06  ; CY2_A_2_BW
OR 2000.15  ; STEP15
AND 22.15  ; MAIN_OK
AND 2000.14  ; STEP14
OUT 2000.15  ; STEP15
TIM 0015 #2  ; TIM_STEP15
; rung 17: DRIVE LIN3
LD 201.13  ; AUTOSIG
AND T0015  ; TIM_STEP15
AND 0.03  ; CY1_FW
AND 0.06  ; CY2_A_2_BW
OR 2002.00  ; STEP16
AND 22.15  ; MAIN_OK
AND 2000.15  ; STEP15
OUT 2002.00  ; STEP16
TIM 0016 #2
; rung 18
LD 201.13  ; AUTOSIG
AND T0016
OR 2002.01  ; STEP17
AND 22.15  ; MAIN_OK
AND 2002.00  ; STEP16
OUT 2002.01  ; STEP17
TIM 0017 #2  ; TIM_S17
; rung 19: LIN1 SET PROGRAM
LD 201.13  ; AUTOSIG
AND 0.03  ; CY1_FW
AND 1.03  ; LIN3_BW
AND T0017  ; TIM_S17
AND P_On
AND P_On
OR 2002.02  ; STEP18
AND 22.15  ; MAIN_OK
AND 2002.01  ; STEP17
OUT 2002.02  ; STEP18
TIM 0018 #2  ; TIM_S18

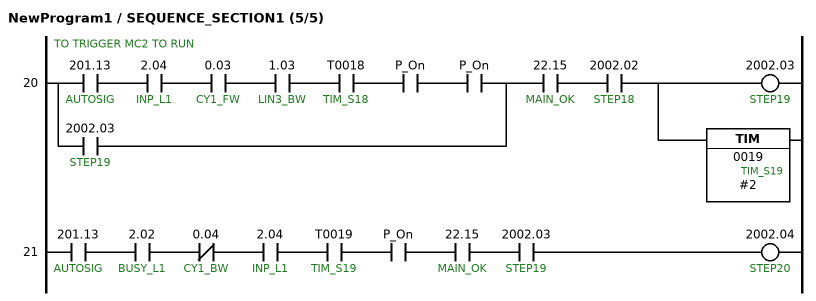
; rung 20: TO TRIGGER MC2 TO RUN
LD 201.13  ; AUTOSIG
AND 2.04  ; INP_L1
AND 0.03  ; CY1_FW
AND 1.03  ; LIN3_BW
AND T0018  ; TIM_S18
AND P_On
AND P_On
OR 2002.03  ; STEP19
AND 22.15  ; MAIN_OK
AND 2002.02  ; STEP18
OUT 2002.03  ; STEP19
TIM 0019 #2  ; TIM_S19
; rung 21
LD 201.13  ; AUTOSIG
AND 2.02  ; BUSY_L1
ANDNOT 0.04  ; CY1_BW
AND 2.04  ; INP_L1
AND T0019  ; TIM_S19
AND P_On
AND 22.15  ; MAIN_OK
AND 2002.03  ; STEP19
OUT 2002.04  ; STEP20

### Section SEQUENCE_SECTION2

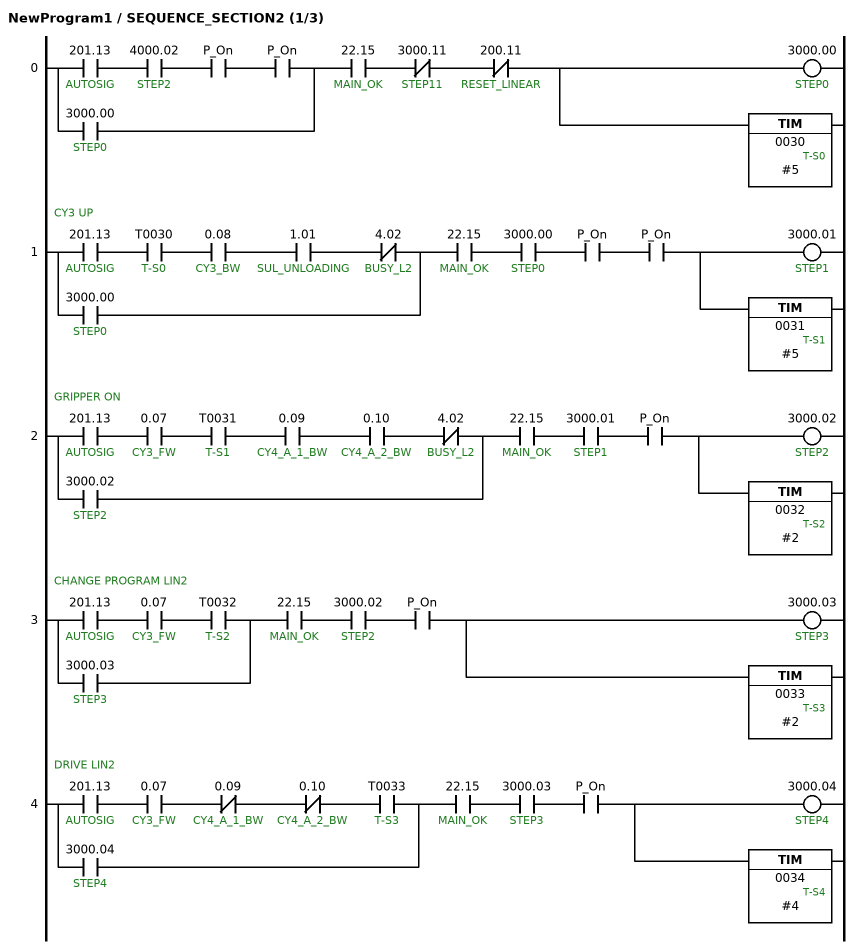
; rung 0
LD 201.13  ; AUTOSIG
AND 4000.02  ; STEP2
AND P_On
AND P_On
OR 3000.00  ; STEP0
AND 22.15  ; MAIN_OK
ANDNOT 3000.11  ; STEP11
ANDNOT 200.11  ; RESET_LINEAR
OUT 3000.00  ; STEP0
TIM 0030 #5  ; T-S0
; rung 1: CY3 UP
LD 201.13  ; AUTOSIG
AND T0030  ; T-S0
AND 0.08  ; CY3_BW
AND 1.01  ; SUL_UNLOADING
ANDNOT 4.02  ; BUSY_L2
OR 3000.00  ; STEP0
AND 22.15  ; MAIN_OK
AND 3000.00  ; STEP0
AND P_On
AND P_On
OUT 3000.01  ; STEP1
TIM 0031 #5  ; T-S1
; rung 2: GRIPPER ON
LD 201.13  ; AUTOSIG
AND 0.07  ; CY3_FW
AND T0031  ; T-S1
AND 0.09  ; CY4_A_1_BW
AND 0.10  ; CY4_A_2_BW
ANDNOT 4.02  ; BUSY_L2
OR 3000.02  ; STEP2
AND 22.15  ; MAIN_OK
AND 3000.01  ; STEP1
AND P_On
OUT 3000.02  ; STEP2
TIM 0032 #2  ; T-S2
; rung 3: CHANGE PROGRAM LIN2
LD 201.13  ; AUTOSIG
AND 0.07  ; CY3_FW
AND T0032  ; T-S2
OR 3000.03  ; STEP3
AND 22.15  ; MAIN_OK
AND 3000.02  ; STEP2
AND P_On
OUT 3000.03  ; STEP3
TIM 0033 #2  ; T-S3
; rung 4: DRIVE LIN2
LD 201.13  ; AUTOSIG
AND 0.07  ; CY3_FW
ANDNOT 0.09  ; CY4_A_1_BW
ANDNOT 0.10  ; CY4_A_2_BW
AND T0033  ; T-S3
OR 3000.04  ; STEP4
AND 22.15  ; MAIN_OK
AND 3000.03  ; STEP3
AND P_On
OUT 3000.04  ; STEP4
TIM 0034 #4  ; T-S4

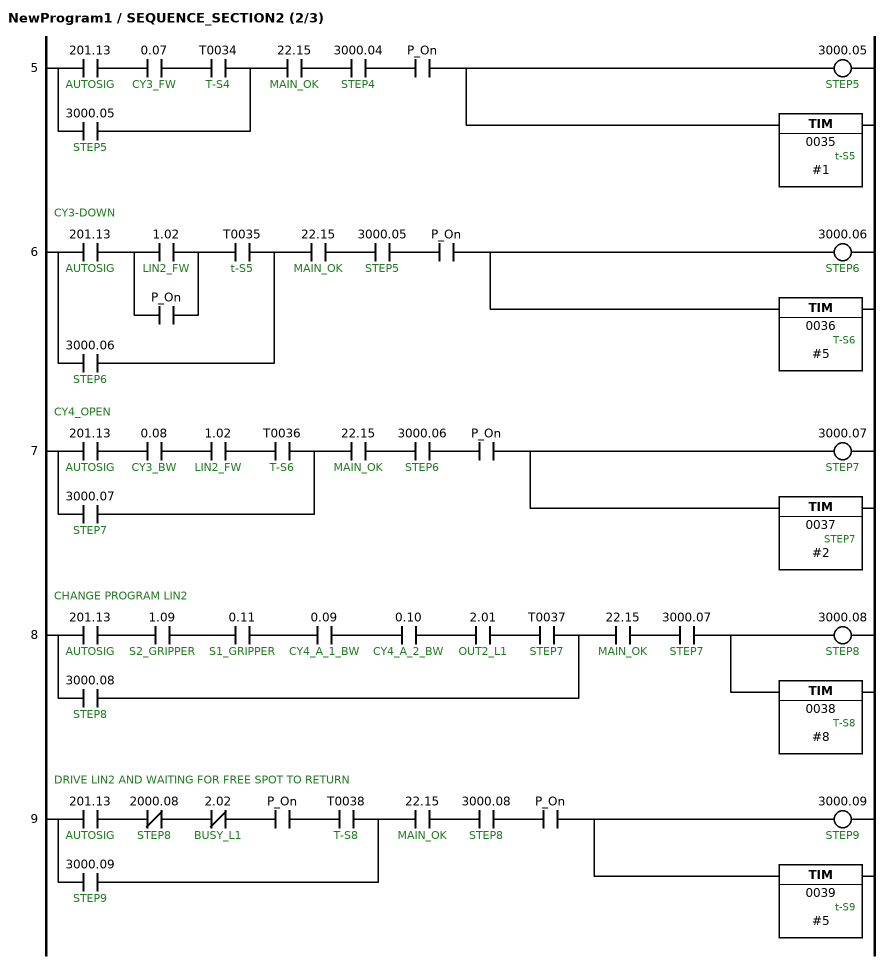
; rung 5
LD 201.13  ; AUTOSIG
AND 0.07  ; CY3_FW
AND T0034  ; T-S4
OR 3000.05  ; STEP5
AND 22.15  ; MAIN_OK
AND 3000.04  ; STEP4
AND P_On
OUT 3000.05  ; STEP5
TIM 0035 #1  ; t-S5
; rung 6: CY3-DOWN
LD 201.13  ; AUTOSIG
LD 1.02  ; LIN2_FW
OR P_On
ANDLD
AND T0035  ; t-S5
OR 3000.06  ; STEP6
AND 22.15  ; MAIN_OK
AND 3000.05  ; STEP5
AND P_On
OUT 3000.06  ; STEP6
TIM 0036 #5  ; T-S6
; rung 7: CY4_OPEN
LD 201.13  ; AUTOSIG
AND 0.08  ; CY3_BW
AND 1.02  ; LIN2_FW
AND T0036  ; T-S6
OR 3000.07  ; STEP7
AND 22.15  ; MAIN_OK
AND 3000.06  ; STEP6
AND P_On
OUT 3000.07  ; STEP7
TIM 0037 #2  ; STEP7
; rung 8: CHANGE PROGRAM LIN2
LD 201.13  ; AUTOSIG
AND 1.09  ; S2_GRIPPER
AND 0.11  ; S1_GRIPPER
AND 0.09  ; CY4_A_1_BW
AND 0.10  ; CY4_A_2_BW
AND 2.01  ; OUT2_L1
AND T0037  ; STEP7
OR 3000.08  ; STEP8
AND 22.15  ; MAIN_OK
AND 3000.07  ; STEP7
OUT 3000.08  ; STEP8
TIM 0038 #8  ; T-S8
; rung 9: DRIVE LIN2 AND WAITING FOR FREE SPOT TO RETURN
LD 201.13  ; AUTOSIG
ANDNOT 2000.08  ; STEP8  // tambahan santo
ANDNOT 2.02  ; BUSY_L1
AND P_On
AND T0038  ; T-S8
OR 3000.09  ; STEP9
AND 22.15  ; MAIN_OK
AND 3000.08  ; STEP8
AND P_On
OUT 3000.09  ; STEP9
TIM 0039 #5  ; t-S9

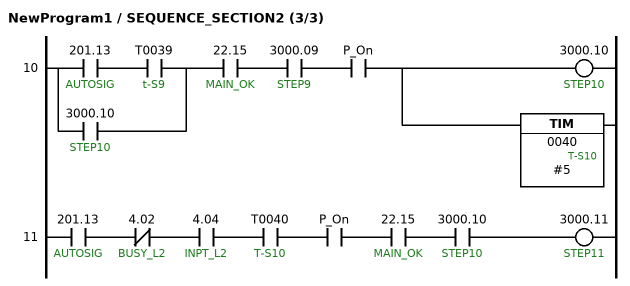
; rung 10
LD 201.13  ; AUTOSIG
AND T0039  ; t-S9
OR 3000.10  ; STEP10
AND 22.15  ; MAIN_OK
AND 3000.09  ; STEP9
AND P_On
OUT 3000.10  ; STEP10
TIM 0040 #5  ; T-S10
; rung 11
LD 201.13  ; AUTOSIG
ANDNOT 4.02  ; BUSY_L2
AND 4.04  ; INPT_L2
AND T0040  ; T-S10
AND P_On
AND 22.15  ; MAIN_OK
AND 3000.10  ; STEP10
OUT 3000.11  ; STEP11

### Section SEQUENCE_MACHINE_2

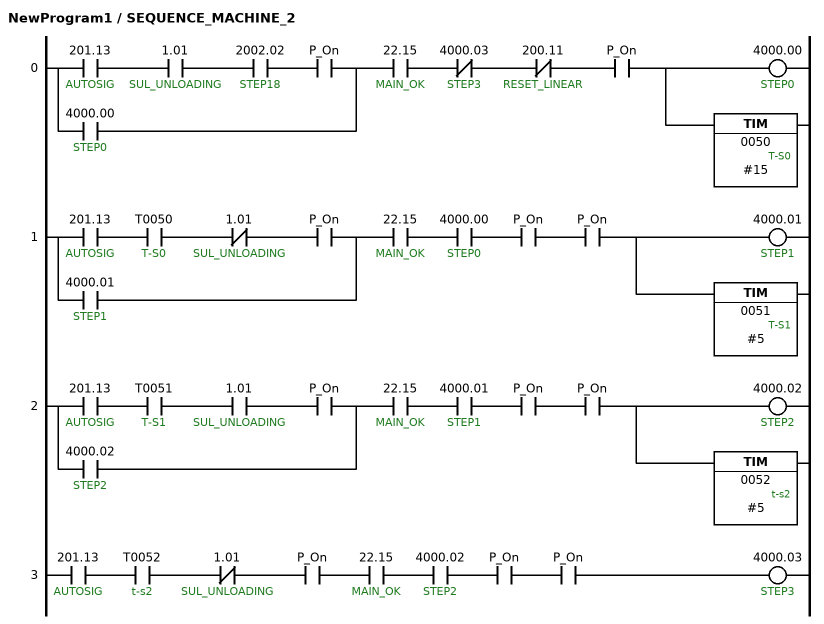
; rung 0
LD 201.13  ; AUTOSIG
AND 1.01  ; SUL_UNLOADING
AND 2002.02  ; STEP18
AND P_On
OR 4000.00  ; STEP0
AND 22.15  ; MAIN_OK
ANDNOT 4000.03  ; STEP3
ANDNOT 200.11  ; RESET_LINEAR
AND P_On
OUT 4000.00  ; STEP0
TIM 0050 #15  ; T-S0
; rung 1
LD 201.13  ; AUTOSIG
AND T0050  ; T-S0
ANDNOT 1.01  ; SUL_UNLOADING
AND P_On
OR 4000.01  ; STEP1
AND 22.15  ; MAIN_OK
AND 4000.00  ; STEP0
AND P_On
AND P_On
OUT 4000.01  ; STEP1
TIM 0051 #5  ; T-S1
; rung 2
LD 201.13  ; AUTOSIG
AND T0051  ; T-S1
AND 1.01  ; SUL_UNLOADING
AND P_On
OR 4000.02  ; STEP2
AND 22.15  ; MAIN_OK
AND 4000.01  ; STEP1
AND P_On
AND P_On
OUT 4000.02  ; STEP2
TIM 0052 #5  ; t-s2
; rung 3
LD 201.13  ; AUTOSIG
AND T0052  ; t-s2
ANDNOT 1.01  ; SUL_UNLOADING
AND P_On
AND 22.15  ; MAIN_OK
AND 4000.02  ; STEP2
AND P_On
AND P_On
OUT 4000.03  ; STEP3

### Section CONVEYOR

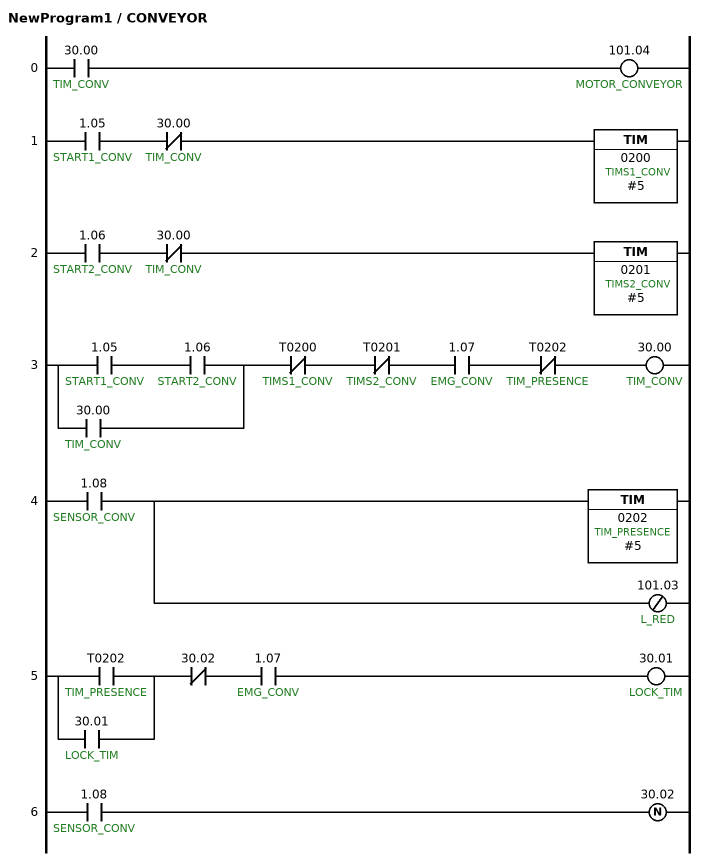
; rung 0
LD 30.00  ; TIM_CONV
OUT 101.04  ; MOTOR_CONVEYOR
; rung 1
LD 1.05  ; START1_CONV
ANDNOT 30.00  ; TIM_CONV
TIM 0200 #5  ; TIMS1_CONV
; rung 2
LD 1.06  ; START2_CONV
ANDNOT 30.00  ; TIM_CONV
TIM 0201 #5  ; TIMS2_CONV
; rung 3
LD 1.05  ; START1_CONV
AND 1.06  ; START2_CONV
OR 30.00  ; TIM_CONV
ANDNOT T0200  ; TIMS1_CONV
ANDNOT T0201  ; TIMS2_CONV
AND 1.07  ; EMG_CONV
ANDNOT T0202  ; TIM_PRESENCE
OUT 30.00  ; TIM_CONV
; rung 4
LD 1.08  ; SENSOR_CONV
TIM 0202 #5  ; TIM_PRESENCE
OUTNOT 101.03  ; L_RED
; rung 5
LD T0202  ; TIM_PRESENCE
OR 30.01  ; LOCK_TIM
ANDNOT 30.02
AND 1.07  ; EMG_CONV
OUT 30.01  ; LOCK_TIM
; rung 6
LD 1.08  ; SENSOR_CONV
DIFD(014) 30.02

### Section END
; rung 0
END(001)